FUNCTION_BLOCK FB_Blinker
VAR_INPUT
	IN	: BOOL;
	PT	: TIME;
END_VAR
VAR_OUTPUT
	Q	: BOOL;
END_VAR
VAR
	TON	: TON;
	TOF	: TOF;
END_VAR

TOF(IN := NOT TON.Q AND IN, PT := PT);
TON(IN := IN AND TOF.Q, PT := PT);

Q := TON.Q;

END_FUNCTION_BLOCK

(* stored: Version 1.1.0.1, ProductVersion 3.1.4024.9
   POU FB_Blinker: Id {70b8d01a-4607-4c4e-9200-cd61d90f7e6c}, SpecialFunc None *)
